INTERFACE I_Component EXTENDS I_Object

METHOD PUBLIC M_OnNotify
VAR_INPUT
	eRequest:		E_Request;
END_VAR
END_METHOD

METHOD PUBLIC M_Request : BOOL
VAR_INPUT
	eRequest:	E_Request;
END_VAR
END_METHOD

PROPERTY PUBLIC P_Event : I_Event
GET
END_GET
END_PROPERTY

PROPERTY PUBLIC P_Info : I_Info
GET
END_GET
END_PROPERTY

PROPERTY PUBLIC P_Observer : I_Observer
GET
END_GET
END_PROPERTY

END_INTERFACE

(* stored: Version 1.1.0.1
   Itf I_Component: Id {84a5f8f6-b81b-4747-a25d-2c3abe61b573}
   Method M_OnNotify: Id {e7af5b28-84d1-47bb-bd50-90d772841703}
   Method M_Request: Id {5bce4574-fbb8-4134-a60e-e5f2d429768c}
   Property P_Event: Id {96ef9ac7-4347-4236-9475-e7c300209edb}
   Get Get: Id {25594f51-5f07-48cf-8274-65c776cd7cf1}
   Property P_Info: Id {a4d97ad8-84af-4536-8ab6-ff3055df9335}
   Get Get: Id {9b0145a7-d929-442e-b904-05f74e6af1bb}
   Property P_Observer: Id {71855be2-d7dd-407c-bfc6-2b33d71db9ac}
   Get Get: Id {06fb4a5b-c62f-47d3-bed0-c50d2d77e5a7} *)
